FUNCTION_BLOCK FB_2003_cookie
VAR_INPUT
	execute: BOOL;
	pos2: LREAL := 2500;
END_VAR
VAR
	TIMERDONE: BOOL;
END_VAR

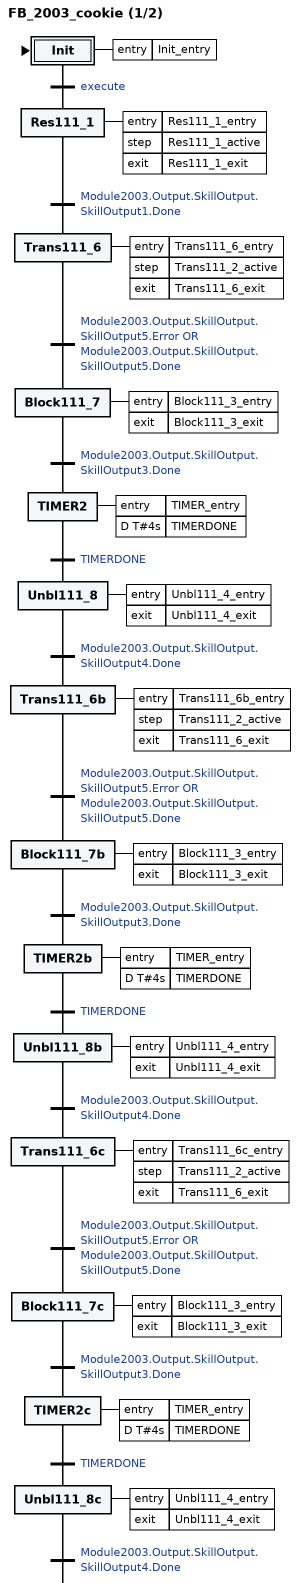
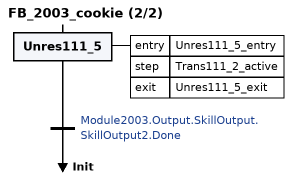
INITIAL_STEP Init:
    Init_entry(P1);  // entry action
END_STEP
TRANSITION FROM Init TO Res111_1
    := execute;
END_TRANSITION
STEP Res111_1:
    Res111_1_entry(P1);  // entry action
    Res111_1_active(N);  // step action
    Res111_1_exit(P0);  // exit action
END_STEP
TRANSITION FROM Res111_1 TO Trans111_6
    := Module2003.Output.SkillOutput.SkillOutput1.Done;
END_TRANSITION
STEP Trans111_6:
    Trans111_6_entry(P1);  // entry action
    Trans111_2_active(N);  // step action
    Trans111_6_exit(P0);  // exit action
END_STEP
TRANSITION FROM Trans111_6 TO Block111_7
    := Module2003.Output.SkillOutput.SkillOutput5.Error OR Module2003.Output.SkillOutput.SkillOutput5.Done;
END_TRANSITION
STEP Block111_7:
    Block111_3_entry(P1);  // entry action
    Block111_3_exit(P0);  // exit action
END_STEP
TRANSITION FROM Block111_7 TO TIMER2
    := Module2003.Output.SkillOutput.SkillOutput3.Done;
END_TRANSITION
STEP TIMER2:
    TIMER_entry(P1);  // entry action
    TIMERDONE(D, T#4s);
END_STEP
TRANSITION FROM TIMER2 TO Unbl111_8
    := TIMERDONE;
END_TRANSITION
STEP Unbl111_8:
    Unbl111_4_entry(P1);  // entry action
    Unbl111_4_exit(P0);  // exit action
END_STEP
TRANSITION FROM Unbl111_8 TO Trans111_6b
    := Module2003.Output.SkillOutput.SkillOutput4.Done;
END_TRANSITION
STEP Trans111_6b:
    Trans111_6b_entry(P1);  // entry action
    Trans111_2_active(N);  // step action
    Trans111_6_exit(P0);  // exit action
END_STEP
TRANSITION FROM Trans111_6b TO Block111_7b
    := Module2003.Output.SkillOutput.SkillOutput5.Error OR Module2003.Output.SkillOutput.SkillOutput5.Done;
END_TRANSITION
STEP Block111_7b:
    Block111_3_entry(P1);  // entry action
    Block111_3_exit(P0);  // exit action
END_STEP
TRANSITION FROM Block111_7b TO TIMER2b
    := Module2003.Output.SkillOutput.SkillOutput3.Done;
END_TRANSITION
STEP TIMER2b:
    TIMER_entry(P1);  // entry action
    TIMERDONE(D, T#4s);
END_STEP
TRANSITION FROM TIMER2b TO Unbl111_8b
    := TIMERDONE;
END_TRANSITION
STEP Unbl111_8b:
    Unbl111_4_entry(P1);  // entry action
    Unbl111_4_exit(P0);  // exit action
END_STEP
TRANSITION FROM Unbl111_8b TO Trans111_6c
    := Module2003.Output.SkillOutput.SkillOutput4.Done;
END_TRANSITION
STEP Trans111_6c:
    Trans111_6c_entry(P1);  // entry action
    Trans111_2_active(N);  // step action
    Trans111_6_exit(P0);  // exit action
END_STEP
TRANSITION FROM Trans111_6c TO Block111_7c
    := Module2003.Output.SkillOutput.SkillOutput5.Error OR Module2003.Output.SkillOutput.SkillOutput5.Done;
END_TRANSITION
STEP Block111_7c:
    Block111_3_entry(P1);  // entry action
    Block111_3_exit(P0);  // exit action
END_STEP
TRANSITION FROM Block111_7c TO TIMER2c
    := Module2003.Output.SkillOutput.SkillOutput3.Done;
END_TRANSITION
STEP TIMER2c:
    TIMER_entry(P1);  // entry action
    TIMERDONE(D, T#4s);
END_STEP
TRANSITION FROM TIMER2c TO Unbl111_8c
    := TIMERDONE;
END_TRANSITION
STEP Unbl111_8c:
    Unbl111_4_entry(P1);  // entry action
    Unbl111_4_exit(P0);  // exit action
END_STEP
TRANSITION FROM Unbl111_8c TO Unres111_5
    := Module2003.Output.SkillOutput.SkillOutput4.Done;
END_TRANSITION
STEP Unres111_5:
    Unres111_5_entry(P1);  // entry action
    Trans111_2_active(N);  // step action
    Unres111_5_exit(P0);  // exit action
END_STEP
TRANSITION FROM Unres111_5 TO Init
    := Module2003.Output.SkillOutput.SkillOutput2.Done;
END_TRANSITION

ACTION Trans111_6_entry:
//TRANSPORTIEREN

Module2003.Input.SkillInput.SkillInput5.Execute := TRUE;
Module2003.Input.SkillInput.SkillInput5.ParameterInput.Parameterinput1.Value := 3000; //X-Position
Module2003.Input.SkillInput.SkillInput5.ParameterInput.Parameterinput2.Value := 80; //Z-Position
Module2003.Input.SkillInput.SkillInput5.ParameterInput.Parameterinput3.Value := 0; //Velocity
Module2003.Input.SkillInput.SkillInput5.ParameterInput.Parameterinput4.Value := 0; //Acceleration
END_ACTION

ACTION Block111_3_exit:
//BLOCKIEREN

Module2003.Input.SkillInput.SkillInput3.Execute := FALSE;
Module2003.Input.SkillInput.SkillInput3.ParameterInput.Parameterinput1.Value := 0; //TaskID
END_ACTION

ACTION Trans111_2_active:

END_ACTION

ACTION Trans111_2_exit:
//TRANSPORTIEREN

Module2003.Input.SkillInput.SkillInput5.Execute := FALSE;
Module2003.Input.SkillInput.SkillInput5.ParameterInput.Parameterinput1.Value := 0; //X-Position
Module2003.Input.SkillInput.SkillInput5.ParameterInput.Parameterinput2.Value := 0; //Z-Position
Module2003.Input.SkillInput.SkillInput5.ParameterInput.Parameterinput3.Value := 0; //Velocity
Module2003.Input.SkillInput.SkillInput5.ParameterInput.Parameterinput4.Value := 0; //Acceleration
END_ACTION

ACTION Block111_3_entry:
//BLOCKIEREN

Module2003.Input.SkillInput.SkillInput3.Execute := TRUE;
Module2003.Input.SkillInput.SkillInput3.ParameterInput.Parameterinput1.Value := 113; //TaskID
END_ACTION

ACTION Unbl111_4_exit:
//unBLOCKIEREN

Module2003.Input.SkillInput.SkillInput4.Execute := FALSE; 
Module2003.Input.SkillInput.SkillInput4.ParameterInput.Parameterinput1.Value := 000; //TaskID
END_ACTION

ACTION Init_entry:
execute := FALSE;
END_ACTION

ACTION Res111_1_active:

END_ACTION

ACTION Trans111_6b_entry:
//TRANSPORTIEREN

Module2003.Input.SkillInput.SkillInput5.Execute := TRUE;
Module2003.Input.SkillInput.SkillInput5.ParameterInput.Parameterinput1.Value := 2600; //X-Position
Module2003.Input.SkillInput.SkillInput5.ParameterInput.Parameterinput2.Value := 80; //Z-Position
Module2003.Input.SkillInput.SkillInput5.ParameterInput.Parameterinput3.Value := 0; //Velocity
Module2003.Input.SkillInput.SkillInput5.ParameterInput.Parameterinput4.Value := 0; //Acceleration
END_ACTION

ACTION Res111_1_exit:
// Reservieren entry
Module2003.Input.SkillInput.SkillInput1.Execute := FALSE;
Module2003.Input.SkillInput.SkillInput1.ParameterInput.Parameterinput1.Value := 0; //TASKID
END_ACTION

ACTION Unres111_5_entry:
//unreserve
Module2003.Input.SkillInput.SkillInput2.Execute := TRUE;
Module2003.Input.SkillInput.SkillInput2.ParameterInput.Parameterinput1.Value := 113; //TaskID
END_ACTION

ACTION Trans111_6c_entry:
//TRANSPORTIEREN

Module2003.Input.SkillInput.SkillInput5.Execute := TRUE;
Module2003.Input.SkillInput.SkillInput5.ParameterInput.Parameterinput1.Value := 3000; //X-Position
Module2003.Input.SkillInput.SkillInput5.ParameterInput.Parameterinput2.Value := 80; //Z-Position
Module2003.Input.SkillInput.SkillInput5.ParameterInput.Parameterinput3.Value := 0; //Velocity
Module2003.Input.SkillInput.SkillInput5.ParameterInput.Parameterinput4.Value := 0; //Acceleration
END_ACTION

ACTION TIMER_entry:
TIMERDONE := FALSE;
END_ACTION

ACTION Unres111_5_exit:
//unreserve
Module2003.Input.SkillInput.SkillInput2.Execute := FALSE;
Module2003.Input.SkillInput.SkillInput2.ParameterInput.Parameterinput1.Value := 0; //TaskID
END_ACTION

ACTION Res111_1_entry:
// Reservieren entry
Module2003.Input.SkillInput.SkillInput1.Execute := TRUE;
Module2003.Input.SkillInput.SkillInput1.ParameterInput.Parameterinput1.Value := 113; //TASKID
END_ACTION

ACTION Trans111_2_entry:
//TRANSPORTIEREN

Module2003.Input.SkillInput.SkillInput5.Execute := TRUE;
Module2003.Input.SkillInput.SkillInput5.ParameterInput.Parameterinput1.Value := 2400; //X-Position
Module2003.Input.SkillInput.SkillInput5.ParameterInput.Parameterinput2.Value := 0; //Z-Position
Module2003.Input.SkillInput.SkillInput5.ParameterInput.Parameterinput3.Value := 300; //Velocity
Module2003.Input.SkillInput.SkillInput5.ParameterInput.Parameterinput4.Value := 100; //Acceleration
END_ACTION

ACTION Trans111_6_exit:
//TRANSPORTIEREN

Module2003.Input.SkillInput.SkillInput5.Execute := FALSE;
Module2003.Input.SkillInput.SkillInput5.ParameterInput.Parameterinput1.Value := 0; //X-Position
Module2003.Input.SkillInput.SkillInput5.ParameterInput.Parameterinput2.Value := 0; //Z-Position
Module2003.Input.SkillInput.SkillInput5.ParameterInput.Parameterinput3.Value := 0; //Velocity
Module2003.Input.SkillInput.SkillInput5.ParameterInput.Parameterinput4.Value := 0; //Acceleration
END_ACTION

ACTION Unbl111_4_entry:
//unBLOCKIEREN

Module2003.Input.SkillInput.SkillInput4.Execute := TRUE; //FALSE weil timer
Module2003.Input.SkillInput.SkillInput4.ParameterInput.Parameterinput1.Value := 112; //TaskID
END_ACTION

END_FUNCTION_BLOCK

(* stored: Version 1.1.0.1, ProductVersion 3.1.0.25
   POU FB_2003_cookie: Id {ffc9393a-a985-445f-ad9e-3d904d52c12d}
   Action Trans111_6_entry: Id {008f24a3-150c-4c4c-a4df-3fc4aa7fd92b}
   Action Block111_3_exit: Id {00bf377e-47e0-49c2-b1cb-43853bf8e8df}
   Action Trans111_2_active: Id {0cc31ef0-0d9b-4ad8-91e3-c6d9e3cda872}
   Action Trans111_2_exit: Id {1840d390-5c49-4447-8ec1-5cea1040f376}
   Action Block111_3_entry: Id {1ae4e92d-1e3c-484a-963e-d3b94b1a56e9}
   Action Unbl111_4_exit: Id {1fcd84e6-6ecb-4d28-9cfd-92adde2969d7}
   Action Init_entry: Id {3776e267-b81b-40b3-b9f2-17f1504bbc3c}
   Action Res111_1_active: Id {47f01fd7-a7f9-497c-b3a1-c5d2614ecf63}
   Action Trans111_6b_entry: Id {5713a8d7-ce65-492f-a8fb-bd0fdc97ba22}
   Action Res111_1_exit: Id {62251339-8c50-4a11-862a-a42530c6d11c}
   Action Unres111_5_entry: Id {7c698e81-1967-463c-9bfc-7ee9dd3d7379}
   Action Trans111_6c_entry: Id {89d0eb5c-bc18-4726-a75c-2863a2c0f7c5}
   Action TIMER_entry: Id {93d900ff-2c8a-4dc1-8f5a-febc7f671e61}
   Action Unres111_5_exit: Id {b9ba22fd-d1e4-473a-aeb3-ac6ddfe8e58b}
   Action Res111_1_entry: Id {c3dae642-a043-4846-be5d-1ea88e52fb8e}
   Action Trans111_2_entry: Id {c6846d1a-55ce-40e9-ad37-bd4def4d3989}
   Action Trans111_6_exit: Id {e291ac4c-eeff-468f-8def-96ceb74670bd}
   Action Unbl111_4_entry: Id {fac7d38e-648c-46aa-a1f1-628b04a94423} *)
